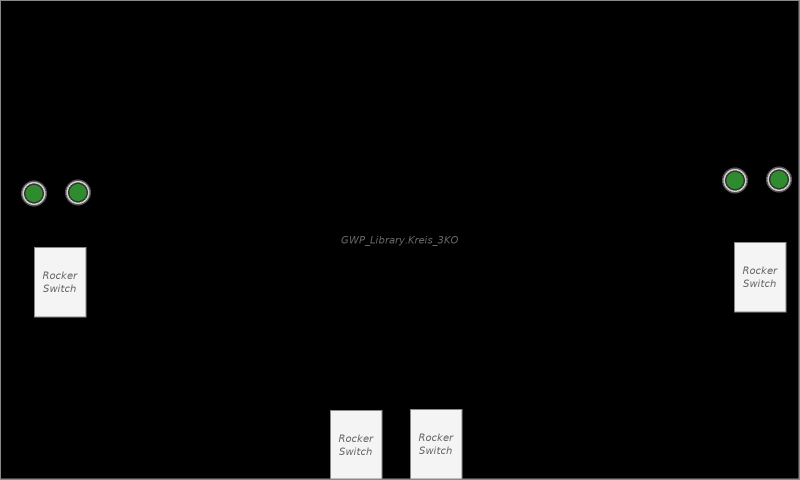
VISUALIZATION Kreis_3KO  // 800x480
    Polygon (903,353)
    Frame (0,0 800x480)
        shows GWP_Library.Kreis_3KO(FB_Kreis_3KO := Main.Kreis_3KO_0, FB_KD := Main.KD_0, FB_VD := Main.VD_0, FB_Init_1 := Main.Init_0)
    Lamp1 (19,178 30x31), variable: MAIN.VD_0.x_BM_Bereit, style: Lamp-Lamp1-Green
    Lamp1 (63,177 30x31), variable: MAIN.VD_0.x_BM_Betrieb, style: Lamp-Lamp1-Green
    RockerSwitch (734,242 52x70), variable: MAIN.KD_0.x_Einschaltbefehl, behaviour: TOGGLE, style: Switch-RockerSwitch-Gray
    RockerSwitch (34,247 52x70), variable: MAIN.VD_0.x_Einschaltbefehl, behaviour: TOGGLE, style: Switch-RockerSwitch-Gray
    RockerSwitch (330,410 52x70), variable: MAIN.einestufe, behaviour: TOGGLE, style: Switch-RockerSwitch-Gray
    RockerSwitch (410,409 52x70), variable: MAIN.zweitestufe, behaviour: TOGGLE, style: Switch-RockerSwitch-Gray
    Lamp1 (720,165 30x31), variable: MAIN.KD_0.x_BM_Bereit, style: Lamp-Lamp1-Green
    Lamp1 (764,164 30x31), variable: MAIN.VD_0.x_BM_Betrieb, style: Lamp-Lamp1-Green
END_VISUALIZATION

(* stored: Version 1.1.0.1, ProductVersion 3.1.4022.6
   Visu Kreis_3KO: Id {daf58c94-67bd-4d25-a781-43ac3830815f} *)
